Yaskawa INFORM job: TESTR2.JBI

/JOB
//NAME TESTR2
///FOLDERNAME INNE
//POS
///NPOS 1,1,0,0,0,0
///TOOL 0
///POSTYPE PULSE
///PULSE
C00000=165479,89885,22654,58298,78947,-15591
BC00000=390128,45261,756517
//INST
///DATE 2023/11/01 18:40
///ATTR SC,RW
///GROUP1 RB1,BS1
NOP
'testr2
MOVJ C00000 BC00000 VJ=100.00
END
